(* IEC 61131-3 sources: com.logicals.lc3.webinar/usRTS_RPMControl_iSOC/src_FB_LIB_SAFE/Numeric/UINT, 8 files *)

(* ---- wADD_UINT_2.iecst ---- *)
NAMESPACE logicals.web.standard
NAMESPACE numeric

/*
 * Function block wrapper for IEC 61131-3 ADD<br>
 * IN1 =  1st value (UINT)<br>
 * IN2 =  2nd value (UINT)<br>
 * OUT = Sum of all input values (UINT)<br>
 */
FUNCTION_BLOCK wADD_UINT_2
	{ vNameAlignment:="center"; altName:="+"; bgColor:="Plum"; width:=40; hideIONames; }
	VAR_INPUT
		IN1 : UINT;
		IN2 : UINT;
	END_VAR
	VAR_OUTPUT
		OUT : UINT;
	END_VAR

	OUT := ADD(IN1:=IN1, IN2:=IN2, ENO=>ENO);
END_FUNCTION_BLOCK

END_NAMESPACE
END_NAMESPACE

(* ---- wADD_UINT_3.iecst ---- *)
NAMESPACE logicals.web.standard
NAMESPACE numeric

/*
 * Function block wrapper for IEC 61131-3 ADD<br>
 * IN1 =  1st value (UINT)<br>
 * IN2 =  2nd value (UINT)<br>
 * IN3 =  3rd value (UINT)<br>
 * OUT = Sum of all input values (UINT)<br>
 */
FUNCTION_BLOCK wADD_UINT_3
	{ vNameAlignment:="center"; altName:="+"; bgColor:="Plum"; width:=40; hideIONames; }
	VAR_INPUT
		IN1 : UINT;
		IN2 : UINT;
		IN3 : UINT;
	END_VAR
	VAR_OUTPUT
		OUT : UINT;
	END_VAR

	OUT := ADD(IN1:=IN1, IN2:=IN2, IN3:=IN3, ENO=>ENO);
END_FUNCTION_BLOCK

END_NAMESPACE
END_NAMESPACE

(* ---- wADD_UINT_4.iecst ---- *)
NAMESPACE logicals.web.standard
NAMESPACE numeric

/*
 * Function block wrapper for IEC 61131-3 ADD<br>
 * IN1 =  1st value (UINT)<br>
 * IN2 =  2nd value (UINT)<br>
 * IN3 =  3rd value (UINT)<br>
 * IN4 =  4th value (UINT)<br>
 * OUT = Sum of all input values (UINT)<br>
 */
FUNCTION_BLOCK wADD_UINT_4
	{ vNameAlignment:="center"; altName:="+"; bgColor:="Plum"; width:=40; hideIONames; }
	VAR_INPUT
		IN1 : UINT;
		IN2 : UINT;
		IN3 : UINT;
		IN4 : UINT;
	END_VAR
	VAR_OUTPUT
		OUT : UINT;
	END_VAR

	OUT := ADD(IN1:=IN1, IN2:=IN2, IN3:=IN3, IN4:=IN4, ENO=>ENO);
END_FUNCTION_BLOCK

END_NAMESPACE
END_NAMESPACE

(* ---- wDIV_UINT.iecst ---- *)
NAMESPACE logicals.web.standard
NAMESPACE numeric

/*
 * Function block wrapper for IEC 61131-3 DIV<br>
 * IN1 =  1st value (UINT)<br>
 * IN2 =  2nd value (UINT)<br>
 * OUT = quotient of IN1 divided by IN2 (UINT)<br>
 */
FUNCTION_BLOCK wDIV_UINT
	{ vNameAlignment:="center"; altName:="/"; bgColor:="Plum"; width:=40; hideIONames; }
	VAR_INPUT
		IN1 : UINT;
		IN2 : UINT;
	END_VAR
	VAR_OUTPUT
		OUT : UINT;
	END_VAR

	OUT := DIV(IN1:=IN1, IN2:=IN2, ENO=>ENO);
END_FUNCTION_BLOCK

END_NAMESPACE
END_NAMESPACE

(* ---- wMUL_UINT_2.iecst ---- *)
NAMESPACE logicals.web.standard
NAMESPACE numeric

/*
 * Function block wrapper for IEC 61131-3 MUL<br>
 * IN1 =  1st value (UINT)<br>
 * IN2 =  2nd value (UINT)<br>
 * OUT = Product of multiplication of all inputs (UINT)<br>
 */
FUNCTION_BLOCK wMUL_UINT_2
	{ vNameAlignment:="center"; altName:="*"; bgColor:="Plum"; width:=40; hideIONames; }
	VAR_INPUT
		IN1 : UINT;
		IN2 : UINT;
	END_VAR
	VAR_OUTPUT
		OUT : UINT;
	END_VAR

	OUT := MUL(IN1:=IN1, IN2:=IN2, ENO=>ENO);
END_FUNCTION_BLOCK

END_NAMESPACE
END_NAMESPACE

(* ---- wMUL_UINT_3.iecst ---- *)
NAMESPACE logicals.web.standard
NAMESPACE numeric

/*
 * Function block wrapper for IEC 61131-3 MUL<br>
 * IN1 =  1st value (UINT)<br>
 * IN2 =  2nd value (UINT)<br>
 * IN3 =  3rd value (UINT)<br>
 * OUT = Product of multiplication of all inputs (UINT)<br>
 */
FUNCTION_BLOCK wMUL_UINT_3
	{ vNameAlignment:="center"; altName:="*"; bgColor:="Plum"; width:=40; hideIONames; }
	VAR_INPUT
		IN1 : UINT;
		IN2 : UINT;
		IN3 : UINT;
	END_VAR
	VAR_OUTPUT
		OUT : UINT;
	END_VAR

	OUT := MUL(IN1:=IN1, IN2:=IN2, IN3:=IN3, ENO=>ENO);
END_FUNCTION_BLOCK

END_NAMESPACE
END_NAMESPACE

(* ---- wMUL_UINT_4.iecst ---- *)
NAMESPACE logicals.web.standard
NAMESPACE numeric

/*
 * Function block wrapper for IEC 61131-3 MUL<br>
 * IN1 =  1st value (UINT)<br>
 * IN2 =  2nd value (UINT)<br>
 * IN3 =  3rd value (UINT)<br>
 * IN4 =  4th value (UINT)<br>
 * OUT = Product of multiplication of all inputs (UINT)<br>
 */
FUNCTION_BLOCK wMUL_UINT_4
	{ vNameAlignment:="center"; altName:="*"; bgColor:="Plum"; width:=40; hideIONames; }
	VAR_INPUT
		IN1 : UINT;
		IN2 : UINT;
		IN3 : UINT;
		IN4 : UINT;
	END_VAR
	VAR_OUTPUT
		OUT : UINT;
	END_VAR

	OUT := MUL(IN1:=IN1, IN2:=IN2, IN3:=IN3, IN4:=IN4, ENO=>ENO);
END_FUNCTION_BLOCK

END_NAMESPACE
END_NAMESPACE

(* ---- wSUB_UINT.iecst ---- *)
NAMESPACE logicals.web.standard
NAMESPACE numeric

/*
 * Function block wrapper for IEC 61131-3 SUB<br>
 * IN1 =  1st value (UINT)<br>
 * IN2 =  2nd value (UINT)<br>
 * OUT = IN1 minus IN2 (UINT)<br>
 */
FUNCTION_BLOCK wSUB_UINT
	{ vNameAlignment:="center"; altName:="-"; bgColor:="Plum"; width:=40; hideIONames; }
	VAR_INPUT
		IN1 : UINT;
		IN2 : UINT;
	END_VAR
	VAR_OUTPUT
		OUT : UINT;
	END_VAR

	OUT := SUB(IN1:=IN1, IN2:=IN2, ENO=>ENO);
END_FUNCTION_BLOCK

END_NAMESPACE
END_NAMESPACE
